// TIA Portal V18 export
// export: Created 2026-01-09T11:23:36.4664933Z, ExportSetting WithDefaults, DisplayName Totally Integrated Automation Portal, DisplayVersion V18 Update 5, DisplayName TIA Portal Openness, DisplayVersion V18 Update 5, DisplayName TIA Portal Teamcenter Gateway, DisplayVersion V18, DisplayName TIA Portal Version Control Interface, DisplayVersion V18, DisplayName SINAMICS Startdrive Advanced, DisplayVersion V18 SP2 Update 1, DisplayName SINAMICS Startdrive G110M, G120, G120C, G120D, G120P, G115D, DisplayVersion V18 SP2 Update 1, DisplayName SINAMICS Startdrive G130, G150, S120, S150, SINAMICS MV, S210, G220, S200, DisplayVersion V18 SP2 Update 1, DisplayName STEP 7 Professional, DisplayVersion V18 Update 5, DisplayName STEP 7 Safety, DisplayVersion V18, DisplayName WinCC Professional, DisplayVersion V18 Update 5
Screen "284_Motor_K2"  1280x800, Number=284, Template=02ManualUnit1
  ScreenLayer "Layer_0"
    Button "btnMenu5" at 512,725 size 128x75  Mode=Text, TextOff="K-电机2 / K-Motor2", TextOn="K-电机2 / K-Motor2"
      on Click: ActivateScreen(Screen name := , Object number := 0)
    FaceplateInstance "Motor_1" at 70,138 size 273x159  FaceplateTypeName=03 FunctionBlocks@$@202 Conveyer_Line@$@202.2 HMI@$@Motor V 0.0.9
      MotorControl := MotorControl_Dev{3}
      InterfacePropertyText "TextName"  Text="K_提升电机 / K_Lifting Motor"
    FaceplateInstance "Motor_2" at 370,138 size 273x159  FaceplateTypeName=03 FunctionBlocks@$@202 Conveyer_Line@$@202.2 HMI@$@Motor V 0.0.9
      MotorControl := MotorControl_Dev{15}
      InterfacePropertyText "TextName"  Text="K_Spare上料电机 / K_SpareLoadingMotor"
    FaceplateInstance "Motor_3" at 670,138 size 273x159  FaceplateTypeName=03 FunctionBlocks@$@202 Conveyer_Line@$@202.2 HMI@$@Motor V 0.0.9
      MotorControl := MotorControl_Dev{16}
      InterfacePropertyText "TextName"  Text="K_Spare下料电机 / K_SpareTakeMotor"
    Button "按钮_9" at 128,725 size 128x75  Mode=Text, PictureOff=向右箭头_0, TextOff="K-气缸1 / K-Cylinder1", TextOn="K-气缸1 / K-Cylinder1"
      on Click: ActivateScreen(Screen name := 280_Cylinder_K1, Object number := 0)
    Button "btnMenu4" at 384,725 size 128x75  Mode=Text, TextOff="K气缸-2 / K-Cylinder2", TextOn="K气缸-2 / K-Cylinder2"
      on Click: ActivateScreen(Screen name := 283_Cylinder_K2, Object number := 0)
    Button "btnMenu6" at 640,725 size 128x75  Mode=Text, TextOff="K-气缸3 / K-Cylinder3", TextOn="K-气缸3 / K-Cylinder3"
      on Click: ActivateScreen(Screen name := 286_Cylinder_K3, Object number := 0)
    Button "btnMenu7" at 896,725 size 128x75  Mode=Text
    Button "btnMenu6_1" at 768,725 size 128x75  Mode=Text, TextOff="K-电机3 / K-Motor3", TextOn="K-电机3 / K-Motor3"
      on Click: ActivateScreen(Screen name := 287_Motor_K3, Object number := 0)
    Button "btnMenu7_1" at 1024,725 size 128x75  Mode=Text
    Button "btnMenu4_1" at 256,725 size 128x75  Mode=Text, TextOff="K-电机1 / K-Motor1", TextOn="K-电机1 / K-Motor1"
      on Click: ActivateScreen(Screen name := 281_Motor_K1, Object number := 0)
